// TwinCAT 3 PLC project PLC1
// ProgramVersion: 3.1.4022.2
// libraries:
//   ERS_CO2 Payload Decoder, * (PXL-Tech)
//   MSC1608 Payload Decoder, * (PXL-Tech)
//   Tc2_BABasic, * (Beckhoff Automation GmbH)
//   Tc2_EnOcean, * (Beckhoff Automation GmbH)
//   Tc2_Standard, * (Beckhoff Automation GmbH)
//   Tc2_System, * (Beckhoff Automation GmbH)
//   Tc2_TcpIp, * (Beckhoff Automation GmbH)
//   Tc2_Utilities, * (Beckhoff Automation GmbH)
//   Tc3_JsonXml, * (Beckhoff Automation GmbH)
//   Tc3_Module, * (Beckhoff Automation GmbH)
//   VisuSymbols,3.5.10.0,System
// project tree:
//   DUTs/ ST_Gwrx.TcDUT, ST_MoteTx.TcDUT, ST_UserData.TcDUT
//   / GlobalTextList.TcGTLO, PlcTask.TcTTO (not stored), Visualization Manager.TcVMO (not stored), VISU_TASK.TcTTO
//   GVLs/ GVL1.TcGVL
//   POUs/ Decoder.TcPOU, DecoderCO2.TcPOU, EnOcean.TcPOU, Json_XML.TcPOU, Lichtsturing.TcPOU, MAIN.TcPOU, Beamercontrol.TcPOU, Tcp_ip.TcPOU
//   VISUs/ Visualization.TcVIS, Visualization_1.TcVIS
// real-time tasks:
//   TASK PlcTask: cycle T#10ms, priority 6, ADS port 350
//   TASK VISU_TASK: cycle T#200000us, priority 30, ADS port 351
//   TASK Standard: cycle T#5ms, priority 20, ADS port 352
// I/O:
//   DEVICE Device 1 (EtherCAT), AmsNetId 5.52.70.129.2.1
//     Term 7 (EK1200) [EK1200-5000 EtherCAT Power supply (2A E-Bus)]
//       Term 8 (EL1008) [EL1008 8Ch. Dig. Input 24V, 3ms]
//       Term 9 (EL2008) [EL2008 8Ch. Dig. Output 24V, 0.5A]
//       Term 10 (EL3062) [EL3062 2Ch. Ana. Input 0-10V]
//       Term 11 (EL4002) [EL4002 2Ch. Ana. Output 0-10V, 12bit]
//       Term 12 (EK1122) [EK1122 2 port EtherCAT junction]
//         Box 13 (BK1150)
//   DEVICE Device 3 (RT-Ethernet Protocol), AmsNetId 5.52.70.129.4.1
//   DEVICE Device 2 (NOV-DP-RAM)
// variable links:
//   EnOcean_Sample_CX9020/EnOcean_Sample_CX9020 Instance <-> Device 1 (EtherCAT)/Term 7 (EK1200)/Term 12 (EK1122)/Box 13 (BK1150)
//     Standard Inputs/.st6581Input/CNODE <-> Term 2 (KL6581)/Channel 1/Input CNODE
//     Standard Inputs/.st6581Input/DB{0..3} <-> Term 2 (KL6581)/Channel 1/Input DB{0..3}  (4 links)
//     Standard Inputs/.st6581Input/ID{0..3} <-> Term 2 (KL6581)/Channel 1/Input ID{0..3}  (4 links)
//     Standard Inputs/.st6581Input/ORG <-> Term 2 (KL6581)/Channel 1/Input ORG
//     Standard Inputs/.st6581Input/STATUS <-> Term 2 (KL6581)/Channel 1/Input STATUS
//     Standard Inputs/.st6581Input/nStatus <-> Term 2 (KL6581)/Channel 1/Status
//     Standard Outputs/.st6581Output/CNODE <-> Term 2 (KL6581)/Channel 1/Output CNODE
//     Standard Outputs/.st6581Output/DB{0..3} <-> Term 2 (KL6581)/Channel 1/Output DB{0..3}  (4 links)
//     Standard Outputs/.st6581Output/ID{0..3} <-> Term 2 (KL6581)/Channel 1/Output ID{0..3}  (4 links)
//     Standard Outputs/.st6581Output/ORG <-> Term 2 (KL6581)/Channel 1/Output ORG
//     Standard Outputs/.st6581Output/STATUS <-> Term 2 (KL6581)/Channel 1/Output STATUS
//     Standard Outputs/.st6581Output/nControl <-> Term 2 (KL6581)/Channel 1/Control

CONFIGURATION PLC1
    RESOURCE PLC ON TwinCAT3
        TASK VISU_TASK(INTERVAL := T#200000us, PRIORITY := 30);
        PROGRAM VisuElems_Visu_Prg WITH VISU_TASK : VisuElems.Visu_Prg;
    END_RESOURCE
END_CONFIGURATION

// ---- DUTs/ST_Gwrx.TcDUT
TYPE ST_Gwrx :
STRUCT
	TimeRec	: STRING;//DATE_AND_TIME ;
	Chan : DINT ;
	Rfch : DINT ;
	Rssi : DINT ;
	Lsnr : REAL ;
END_STRUCT
END_TYPE

// ---- DUTs/ST_MoteTx.TcDUT
TYPE ST_MoteTx :
STRUCT
	Freq	: DINT ;
	Modu	: STRING(20);
	Datr	: STRING(20);
	Codr	: STRING(20);
END_STRUCT
END_TYPE

// ---- DUTs/ST_UserData.TcDUT
TYPE ST_UserData :
STRUCT
	SeqNo	: DINT;
	Port	: DINT;
	Payload	: STRING;
	Payload2: DINT;
	MoteTx	: ST_MoteTx;
	Gwrx : ST_Gwrx;
END_STRUCT
END_TYPE

// ---- GVLs/GVL1.TcGVL
VAR_GLOBAL
	
//lichtsturing
LichtenRAAMKANT AT %Q*: BOOL;
LichtenDEURKANT AT %Q*: BOOL;

AanwezigheidsdetectorRAAMKANT AT %I*: BOOL;
AanwezigheidsdetectorDEURKANT AT %I*: BOOL;

LichtsterkteDEUR AT %I*: INT;
LichtsterkteDEUR2 AT %I*: INT;
LichtsterkteBORD AT %I*: INT;
lichtsterkteBORD2 AT %I*: INT;
LINKERKNOP AT %I* : BOOL;
RECHTERKNOP AT %I* : BOOL;


//beamer & projectorschermsturing

BeamerAANKNOP AT %I* : BOOL;
BeamerUITKNOP AT %I* : BOOL;
Projectorscherm AT %Q* : BOOL;



socketconnectknop AT %I* : BOOL;
socketsendknop AT %I* : BOOL;



//raamsturing


stKL6581            : STR_KL6581;


//Lora
	sDatastring: STRING(500);
	
	Moteeui			: STRING;
	Appeui			: STRING;
	UserData		: ST_UserData;
	PayloadDecoded	: STRING;

	PayloadLength	: DINT;
	PayloadData		: ARRAY[1..100] OF BYTE;
	NullByte		: BYTE := 0;


END_VAR

// ---- POUs/Lichtsturing.TcPOU
PROGRAM Lichtsturing

 VAR PERSISTENT
	relaisstandDEUR : BOOL := FALSE;
 	relaisstandRAAM : BOOL := FALSE;
 
 
 END_VAR
 
 
VAR
	timer1: TOF;
	timer2: TOF;
	TP1: TP;
	TP2 : TP;
	TP3 : TP;
	TP4 : TP;
	TP5 :TP;
	TP6 : TP;
	
	bewegingraam : BOOL;
	bewegingdeur : BOOL;
	relaisstandDEUR_nieuw : BOOL := FALSE;
	lichtstand2 : BOOL;
	Lichtstand_Prev2: BOOL;
	Lichtstand_Prev: BOOL;
	LichtstatusDEUR : BOOL;
	LichtstatusBORD : BOOL;
	
	

	TONBOOL: BOOL;
	TON1: TON;
	rtrigger: R_TRIG;
	rtrigger2: R_TRIG;
	rtrigger3: R_TRIG;
	rtrigger4: R_TRIG;
	LINKERKNOPULS: BOOL;
	RECHTERKNOPPULS: BOOL;
	
	lichtsterktedeurBerekening: INT := 30000;
	lichtsterkteraamBerekening: INT := 15000;
	fblicht: FB_Light;
	fblicht2 : FB_light;
	relaisstandraam_nieuw: BOOL;
END_VAR

timer1(IN:=gvl1.AanwezigheidsdetectorRAAMKANT, PT:= T#300S, Q=>bewegingraam, ET=> );
timer2(IN:=gvl1.AanwezigheidsdetectorDEURKANT, PT:= T#300S, Q=>bewegingdeur , ET=> );



fblicht(bOn:= (LichtsterkteDEUR + LichtsterkteDEUR2 < lichtsterktedeurBerekening AND bewegingdeur = TRUE), 
bOff:= NOT (LichtsterkteDEUR + LichtsterkteDEUR2 < lichtsterktedeurBerekening AND bewegingdeur = TRUE), 
bToggle:=RECHTERKNOP, bLight=> relaisstandDEUR_nieuw);

IF (relaisstandDEUR = NOT relaisstandDEUR_nieuw) THEN
	TP2.IN := TRUE;
	relaisstandDEUR := relaisstandDEUR_nieuw;
ELSE
	TP2.IN := FALSE;
END_IF


TP2( PT:=T#50MS , Q => GVL1.LichtenDEURKANT);


fblicht2(bOn:= (LichtsterkteBORD + lichtsterkteBORD2 < lichtsterkteraamBerekening AND bewegingraam = TRUE), 
bOff:= NOT (LichtsterkteBORD + lichtsterkteBORD2 < lichtsterkteraamBerekening AND bewegingraam = TRUE), 
bToggle:=LINKERKNOP, bLight=> relaisstandraam_nieuw);

IF (relaisstandraam = NOT relaisstandraam_nieuw) THEN
	TP1.IN := TRUE;
	relaisstandraam := relaisstandraam_nieuw;
ELSE
	TP1.IN := FALSE;
END_IF


TP1( PT:=T#50MS , Q => GVL1.LichtenRAAMKANT);

END_PROGRAM

// ---- POUs/Decoder.TcPOU
PROGRAM Decoder
VAR
 	FB_Decoder : MCS1608_Payload_Decoder;
    //GenSens
 	Status     			:BYTE;      // Content Depends on Message ID == for future use
	BaromBar			:REAL;      // Air Pressure in mBar
	Temp1   			:REAL;     	// in 0,01 degC
	Humidity   			:BYTE;      // Relative Humidity in %
	LevelX     			:SINT;      // Inverse Sinus of Spirit Level in Deg X-Direction -128 = -90 Degr .. +127 = +90 Degr
	LevelY     			:SINT;      // Inverse Sinus of Spirit Level in Deg Y-Direction -128 = -90 Degr .. +127 = +90 Degr
	LevelZ     			:SINT;      // Inverse Sinus of Spirit Level in Deg Z-Direction -128 = -90 Degr .. +127 = +90 Degr
	VibAmp     			:USINT;     // Amplitude of Vibration Detected == Future
	VibFreq    			:USINT;     // Approx. Frequency of Vibration Detected in Hz == Future



	//Tracking
	Start				:BOOL;// Start Message
	Moving				:BOOL;// Object Moving
	Stop				:BOOL;// Object Stopped
	Vibr				:BOOL;// Vibration Detected
	Temp2				:REAL;// Temperature in 0,01 degC
	GPSFixAge			:BYTE;// bit 0..7 = Age of last GPS Fix in Minutes,
	SatCnt_HiLL			:BYTE;// bit 0..4 = SatInFix, bit5 Latitude 25 bit 6,7 = Longitude 25,26
	Lat					:REAL;
	Lon					:REAL;
	
	//Alarm
	GravRotAl		:BOOL;	// Gravity Rotation Detected
	MagRot			:BOOL;	// Magnetic Rotation Detected
	MotAlarm		:BOOL;	// Motion Alarm Detected
	GeoFenceAl		:BOOL;	// GeoFence Violation Detected
	VibrAl			:BOOL;	// Vibration Alarm Detected
	ShockAl			:BOOL;	// Shock Alarm (future use)
	DigIn1Al		:BOOL;	// Digin1 Alarm Detected
	DigIn2Al		:BOOL;	// Digin2 Alarm Detected
	Temp			:REAL;	// Temperature in 0,01 Celcius
	Hum				:BYTE;	// Relative Humidity in %
	BaromBar2		:REAL;	// Air Pressure in Mbar
	
	Alarm1 : Alarm; 
END_VAR

FB_Decoder(dataString := PayloadDecoded);

CASE FB_Decoder.MsgID OF 
	FB_Decoder.ID_Tracking:
		//Start := FB_Decoder.Tracking.Start;
		Moving := FB_Decoder.Tracking.Moving;
		Stop := FB_Decoder.Tracking.Stop;
		Vibr := FB_Decoder.Tracking.Vibr;
		Temp2 := FB_Decoder.Tracking.Temp;
		GPSFixAge := FB_Decoder.Tracking.GPSFixAge;
		SatCnt_HiLL	:= FB_Decoder.Tracking.SatCnt_HiLL;
		Lat	:= FB_Decoder.Tracking.Lat;
		Lon	:= FB_Decoder.Tracking.Lon;
	FB_Decoder.ID_Alarm:
		Alarm1.MotAlarm := FB_Decoder.Alarm.MotAlarm;
	FB_Decoder.ID_GenSens:
		Status := FB_Decoder.GenSens.Status;
		BaromBar := FB_Decoder.GenSens.BaromBar;
		Temp := FB_Decoder.GenSens.Temp;
		Humidity := FB_Decoder.GenSens.Humidity;
		LevelX := FB_Decoder.GenSens.LevelX;
		LevelY := FB_Decoder.GenSens.LevelY;
		LevelZ := FB_Decoder.GenSens.LevelZ;
		VibAmp := FB_Decoder.GenSens.VibAmp;
		VibFreq := FB_Decoder.GenSens.VibFreq;
END_CASE

END_PROGRAM

// ---- POUs/DecoderCO2.TcPOU
PROGRAM DecoderCO2
VAR
	FB_Decoder : ERS_CO2_PayloadDecoder;
	
	Temperature 	: REAL;		//Temp -3276.8°C - 3276.7°C
	Humidity 		: BYTE;		//Humidity 0-100%
	X 				: REAL;		//Acceleration X -128 --> 127 +/-63 = 1G
	Y 				: REAL;		//Acceleration Y -128 --> 127 +/-63 = 1G
	Z 				: REAL;		//Acceleration Z -128 --> 127 +/-63 = 1G
	Light 			: WORD; 	//Light 0 - 65535 Lux
	Motion 			: BYTE;		//No of motion 0-255
	Co2				: WORD;		//Co2 0-65535 ppm 
	Vdd				: WORD;		//VDD 0-65535mV
	Analog1			: WORD;		//VDD 0-65535mV
	Lat				: DWORD;	//Latitude binary
	Lon				: DWORD;	//Longitude binary
	Pulse1			: WORD;		//Relative pulse count
	pulseAbs		: DWORD;	//no 0 - 0xFFFFFFFF
	ExternalTemp	: REAL;		//External temp -3276.5C-->3276.5C
	Digital			: BYTE;		//Value 1 or 0
	Distance		: WORD;		//Distance in mm
	AccMotion		: BYTE;		//Number of vibration/motion
	IrInternalTemp	: REAL;		//Internal temp -3276.5C - 3276.5C
	IrExternalTemp	: REAL;		//External temp -3276.5C - 3276.5C
	Occupancy		: BYTE;		//Data
	Waterleak		: BYTE;		//Data 0-255
	Pressure		: REAL;		//Pressure data(hPa)
	SoundPeak		: BYTE;		//Sound peak
	SoundAvg		: BYTE;		//Sound average
	Pulse2			: WORD;		//0 - 0xFFFF
	PulseAbs2		: DWORD;	//no 0 - 0xFFFFFFFF
	Analog2			: WORD;		//Voltage in mV
	ExternalTemp2	: REAL;		//External temp2 -3276.5C - 3276.5C
END_VAR

FB_Decoder(dataString := PayloadDecoded);

		Temperature 	:= FB_Decoder.Temperature;
		Humidity 		:= FB_Decoder.Humidity;
		X 				:= FB_Decoder.X;
		Y 				:= FB_Decoder.Y;
		Z 				:= FB_Decoder.Z;
		Light 			:= FB_Decoder.Light;		
		Motion 			:= FB_Decoder.Motion;
		Co2				:= FB_Decoder.Co2; 
		Vdd				:= FB_Decoder.Vdd;
		Analog1			:= FB_Decoder.Analog1;
		Lat				:= FB_Decoder.Lat;
		Lon				:= FB_Decoder.Lon;
		Pulse1			:= FB_Decoder.Pulse1;
		pulseAbs		:= FB_Decoder.pulseAbs;
		ExternalTemp	:= FB_Decoder.ExternalTemp;
		Digital			:= FB_Decoder.Digital;
		Distance		:= FB_Decoder.Distance;
		AccMotion		:= FB_Decoder.AccMotion;
		IrInternalTemp	:= FB_Decoder.IrInternalTemp;
		IrExternalTemp	:= FB_Decoder.IrExternalTemp;
		Occupancy		:= FB_Decoder.Occupancy;
		Waterleak		:= FB_Decoder.Waterleak;
		Pressure		:= FB_Decoder.Pressure;
		SoundPeak		:= FB_Decoder.SoundPeak;
		SoundAvg		:= FB_Decoder.SoundAvg;
		Pulse2			:= FB_Decoder.Pulse2;
		PulseAbs2		:= FB_Decoder.PulseAbs2;
		Analog2			:= FB_Decoder.Analog2;
		ExternalTemp2	:= FB_Decoder.ExternalTemp2;

END_PROGRAM

// ---- POUs/EnOcean.TcPOU
PROGRAM EnOcean

VAR
	
FBRECEX: FB_Rec_Teach_In_Ex;


rxD: FB_KL6581;
fbkl6581: FB_KL6581;
	
stKL6581_in AT %I* : KL6581_Input;
stKL6581_out AT %Q* : KL6581_Output; 


testvar2: INT;
	generic1: FB_Rec_1BS;
	generic2: FB_Rec_1BS;
END_VAR



VAR_INPUT 
	//84246605
	//84246441
//fbkl6581
bInit             : BOOL;
nIdx              : USINT := 2;


//FBRECEX
	
bStart            : BOOL;
byNode            : BYTE;
str_KL6581        : STR_KL6581;
DeviceID : DWORD := 0;
testvar : INT := 0;

dw_ID                  : DWORD;

END_VAR



VAR_OUTPUT
	

bReady            : BOOL;
bBusy             : BOOL;
bError            : BOOL;
iErrorID          : E_KL6581_Err;

	

	
bLearnType        : BOOL;
by_Node           : BYTE;

str_Teach_In      : STR_Teach;
bReceive          : BOOL := TRUE;
bReceive2         : BOOL := TRUE;


raam1open          : BOOL;
raam1gesloten          : BOOL;
bLRN            : BOOL;

raam2open         : BOOL;
raam2gesloten         : BOOL;
bLRN2           : BOOL;


END_VAR


fbkl6581(
	bInit:= TRUE , 
	nIdx:= nIdx, 
	bReady=> bReady, 
	bBusy=> bBusy, 
	bError=> bError, 
	iErrorID=> iErrorID, 
	str_KL6581=> str_KL6581, 
	
	stKL6581_in:= stKL6581_in, 
	stKL6581_out:= stKL6581_out);
	
	

FBRECEX(
	bStart:= TRUE, 
	byNode:= 0,
	str_KL6581:= str_KL6581, 
	bLearnType=> , 
	by_Node=>by_node, 
	dw_ID=>DeviceID, 
	str_Teach_In=> str_Teach_In , );
	//bReceive=>bReceive );
	
	
	generic1(
	str_KL6581:= str_KL6581  , 
	byNode:= 0, 
	dw_ID:= 84246605, 
	bOpen=> raam1open, 
	bClose=> raam1gesloten, 
	bLRN=> bLRN2, 
	by_Node=> , 
	bReceive=>bReceive );
	
	generic2(
	str_KL6581:= str_KL6581  , 
	byNode:= 0, 
	dw_ID:= 84246441, 
	bOpen=> raam2open, 
	bClose=> raam2gesloten, 
	bLRN=> bLRN, 
	by_Node=> , 
	bReceive=> bReceive2);

END_PROGRAM

// ---- POUs/Json_XML.TcPOU
PROGRAM Json_XML
VAR
	
	//sJsontest		: STRING(500) := '{"rx": {"moteeui": "00-59-ac-00-00-15-10-ee", "appeui": "0000000000000000", "userdata": {"seqno": 122, "port": 1, "payload": "MDIwMDA1YWUwOTdhMzYwMDAwZmEwMDAwMDAwMDAwMDA=", "motetx": {"freq": 868300000, "modu": "LoRa", "datr": "SF8BW125", "codr": "4/5"}}, "gwrx":  [{"time": "2017-10-17 12:34:53", "chan": 4, "rfch": 0, "rssi": -34, "lsnr": 11.800000000000001}]}}';	
	//sJsontest		: STRING(500) := '{"rx": {"moteeui": "00-59-ac-00-00-15-10-ee", "appeui": "0000000000000000", "userdata": {"seqno": 122, "port": 1, "payload": "MDIwMDA1YWUwOTdhMzYwMDAwZmEwMDAwMDAwMDAwMDA=", "motetx": {"freq": 868300000, "modu": "LoRa", "datr": "SF8BW125", "codr": "4/5"}}, "gwrx": [{"time": "2017-10-17 12:34:53", "chan": 4, "rfch": 0, "rssi": -34, "lsnr": 11.800000000000001}]}}';	
	
	x : DINT;
	g : STRING;
	fbJson			: FB_JsonDomParser;
	JsonDoc			: SJsonValue;
	Json_St1		: SJsonValue;
	JSon_St2		: SJsonValue; 
	JSon_St3		: SJsonValue;
	JSon_St4		: SJsonValue;
	JSon_St5		: SJsonValue;
	JSon_St6		: SJsonValue;
	Stringdata		: STRING;
	
	i: INT;
END_VAR

FOR i := 0 TO 498 DO										//Forloop doorloop elk teken appart
	IF sDatastring[i] = 91 OR sDatastring[i] = 93 THEN		//ALs er een vierkante haak  voor komt
		sDatastring[i] := 32;								//Zal het door een spatie gewijzigd worden
	END_IF
END_FOR

JsonDoc := fbJson.ParseDocument(sDatastring);

// rx
Json_St1 := fbJson.FindMember(jsonDoc, 'rx');			

	// moteeui 
	JSon_St2 := fbJson.FindMember(Json_St1, 'moteeui');
	Moteeui := fbJson.GetString(JSon_St2);

	// appeui	
	JSon_St2 := fbJson.FindMember(Json_St1, 'appeui');
	Appeui := fbJson.GetString(JSon_St2);

	// userdata
	JSon_St2 := fbJson.FindMember(Json_St1, 'userdata');

		// seqno
		JSon_St3 := fbJson.FindMember(Json_St2, 'seqno');
		UserData.SeqNo := fbJson.GetInt(JSon_St3);

		// port
		JSon_St3 := fbJson.FindMember(Json_St2, 'port');
		UserData.Port := fbJson.GetInt(JSon_St3);

		// payload
		JSon_St3 := fbJson.FindMember(Json_St2, 'payload');
		UserData.Payload := fbJson.GetString(JSon_St3);
		PayloadLength:= fbJson.GetBase64(JSon_St3, ADR(PayloadData), SIZEOF(PayloadData));
		Memcpy(ADR(PayloadDecoded), ADR(PayloadData), PayloadLength);
		Memcpy(ADR(PayloadDecoded)+PayloadLength, adr(NullByte), 1);

		// motetx
		JSon_St3 := fbJson.FindMember(Json_St2, 'motetx');

			// freq
			JSon_St4 := fbJson.FindMember(Json_St3, 'freq');
			UserData.MoteTx.Freq := fbJson.GetInt(JSon_St4);

			// modu
			JSon_St4 := fbJson.FindMember(Json_St3, 'modu');
			UserData.MoteTx.Modu := fbJson.GetString(JSon_St4);

			// datr
			JSon_St4 := fbJson.FindMember(Json_St3, 'datr');
			UserData.MoteTx.Datr := fbJson.GetString(JSon_St4);

			// codr
			JSon_St4 := fbJson.FindMember(Json_St3, 'codr');
			UserData.MoteTx.Codr := fbJson.GetString(JSon_St4);

		// gwrx
		JSon_St5 := fbJson.FindMember(Json_St1, 'gwrx');
		Stringdata := fbJson.GetString(JSon_St5);

		// seqno
		JSon_St6 := fbJson.FindMember(Json_St5, 'time');
		UserData.gwrx.TimeRec  := fbJson.GetString(JSon_St6);

END_PROGRAM

// ---- POUs/MAIN.TcPOU
PROGRAM MAIN
VAR
END_VAR

Lichtsturing();
EnOcean();
Beamercontrol();
Tcp_ip();

END_PROGRAM

// ---- POUs/Beamercontrol.TcPOU
PROGRAM Beamercontrol



VAR
	
	fbsocketsend: FB_SocketSend;
	bconnect AT %I* : BOOL;
	test : int;
	clientserver: FB_ClientServerConnection;


	
	Beamerstand: LINT;
END_VAR


VAR_INPUT

       
nMode           : DWORD := 16#8000000;



 
BeamerON    : LINT := 16#020000000002;


BeamerOFF 	: LINT := 16#020100000003;
					  

beamerINPUTCHANGE : LINT :=16#020300000201060E;


	
	 


      	sSrvNetId       : T_AmsNetId := '5.52.70.129.1.1';
	  
        sRemoteHost     : STRING(15) := '192.168.0.102';
        nRemotePort     : UDINT := 7142;
        bExecute                : BOOL;
        tTimeout                : TIME := T#45S;
		tReconnect      : TIME := T#45S;(*!!!*)
		

//socketsend       
               
        cbLen           : UDINT;                        
        pSrc            : DWORD;    
		            
           
END_VAR  

VAR_OUTPUT
        bBusy           : BOOL;
        bError          : BOOL;
        nErrId          : UDINT;
		nErrId2          : UDINT;
        hSocket        : T_HSOCKET;
		eState          : E_SocketConnectionState := eSOCKET_DISCONNECTED;
		
	
END_VAR

clientserver(
	sSrvNetID:= '', 
	nMode:=CONNECT_MODE_ENABLEDBG , 
	sRemoteHost:= sremoteHost , 
	nRemotePort:= nremoteport, 
	bEnable:= bconnect, 
	tReconnect:= tReconnect, 
	bBusy=> bBusy, 
	bError=> berror,
	nErrId=>nErrId , 
	hSocket=>hsocket , 
	eState=> eState);
	
	IF BeamerAANKNOP = TRUE THEN
		bExecute := TRUE;
		Beamerstand := BeamerON;
ELSE
	IF BeamerUITKNOP = TRUE THEN
		bExecute := TRUE;
		Beamerstand := BeamerOFF;
	ELSE
		bExecute := FALSE;
		Beamerstand := 0;
	END_IF
	END_IF
	
fbsocketsend(
	sSrvNetId:='' , 
	hSocket:= clientserver.hSocket, 
	cbLen:= 50, 
	pSrc:= ADR(Beamerstand), 
	bExecute:= bexecute , 
	tTimeout:=tTimeout , 
	bBusy=> bBusy , 
	bError=> bError, 
	nErrId=> nErrId2);

END_PROGRAM

// ---- POUs/Tcp_ip.TcPOU
PROGRAM Tcp_ip
VAR
	bConnect: BOOL;
	bRecieve: BOOL;
	FB_create: FB_SocketUdpCreate;
	FB_Recieve: FB_SocketUdpReceiveFrom;
	FB_close: FB_SocketClose;
	data : ARRAY[0..500] OF BYTE;
END_VAR

FB_create(
	sSrvNetId:= , 							//Lokaal netwerk (mag leeg blijven)
	sLocalHost:= '192.168.0.104', 			//Eigen ip van de PC en ingesteld in de gateway
	nLocalPort:= 811,						//Ingesteld op de gateway
	bExecute:= bConnect,					//Trigger voor functieblok
	tTimeout:= T#45S);
	

FB_Recieve(
	sSrvNetId:= , 									//Lokaal netwerk (mag leeg blijven)
	hSocket:= FB_create.hSocket,					 
	cbLen:= SIZEOF(data), 							//Kijkt naar de lengte van het bericht
	pDest:= ADR(data), 								//Plaat waar de het bericht wordt opgeslaan
	bExecute:= NOT FB_recieve.bBusy AND bRecieve, 	//Trigger voor functieblok
	tTimeout:= T#45S);
	
FB_close(
	sSrvNetId:= , 							//Lokaal netwerk (mag leeg blijven)
	hSocket:= FB_create.hSocket, 			
	bExecute:= NOT bConnect, 				//Sluiten van de connectie 
	tTimeout:= T#45S);
	
IF FB_Recieve.nRecBytes > 0 THEN 										//Dit gebuert op het moment dat er data binnenkomt
	memcpy(ADR(sDatastring),ADR(data),FB_Recieve.nRecBytes);			//Het bericht zal worden opgeslaan in Datastring
	memcpy(ADR(sDatastring) + FB_Recieve.nRecBytes,ADR(NullByte),1);	//Nullbyte word gedetecteerd stoppen met bericht plaatsen
	Json_XML();															//Oproepen POU Json_XML - MOET hier anders bluescreen
	Decoder();
	DecoderCO2();															//Oproepen POU Decoder  - MOET hier anders bluescreen
END_IF

END_PROGRAM

// ---- GlobalTextList.TcGTLO
TEXTLIST GlobalTextList
  820 = 'Bar : %d'
  42 = 'Beamer OFF'
  198 = 'Beamer ON'
  817 = 'Close'
  831 = 'Conection'
  492 = 'Connect'
  830 = 'Create'
  833 = 'Datum/Tijd : %s'
  787 = 'Deurkant'
  828 = 'Error'
  822 = 'Humidity : %d %'
  823 = 'Level x : %d'
  824 = 'Level y : %d'
  825 = 'Level z : %d'
  818 = 'Mesage ID : %d'
  816 = 'Payload : %s'
  774 = 'Raamkant'
  815 = 'Recieve'
  829 = 'Sensor ID : %s'
  819 = 'Status : %d'
  821 = 'Temp : %.2f °c'
  832 = 'Type sensor : '
  826 = 'VibAmp : %d'
  827 = 'VidFreq : %d'
END_TEXTLIST

// ---- VISUs/Visualization.TcVIS
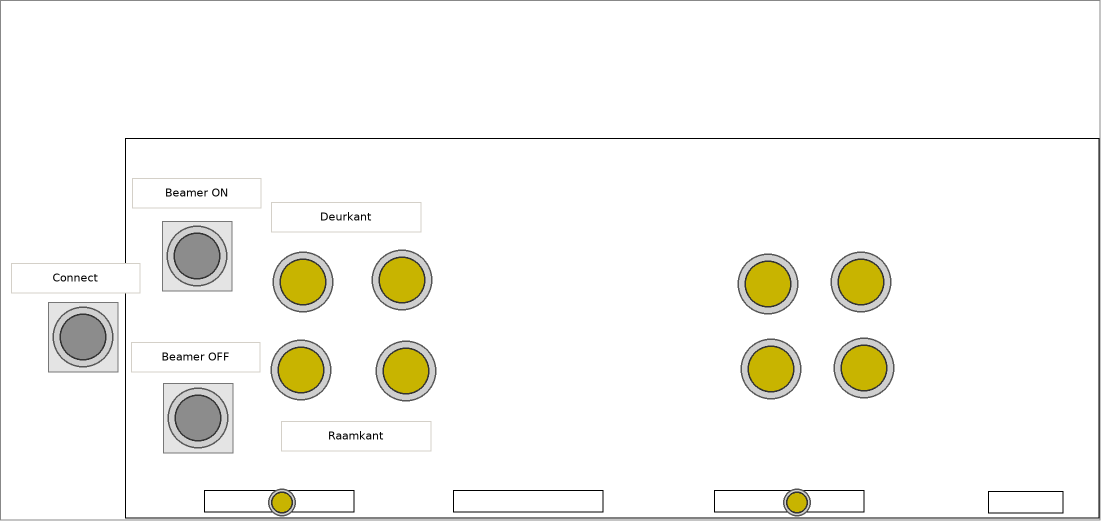
VISUALIZATION Visualization  // 1101x521
    Rectangle (125,138 974x380)
    Lamp1 (268,247 70x70), variable: Lichtsturing.relaisstandDEUR, style: Lamp-Lamp1-Yellow
    Lamp1 (367,245 70x70), variable: Lichtsturing.relaisstandDEUR, style: Lamp-Lamp1-Yellow
    Lamp1 (733,249 70x70), variable: Lichtsturing.relaisstandDEUR, style: Lamp-Lamp1-Yellow
    Lamp1 (826,247 70x70), variable: Lichtsturing.relaisstandDEUR, style: Lamp-Lamp1-Yellow
    Lamp1 (266,335 70x70), variable: Lichtsturing.relaisstandRAAM, style: Lamp-Lamp1-Yellow
    Lamp1 (371,336 70x70), variable: Lichtsturing.relaisstandRAAM, style: Lamp-Lamp1-Yellow
    Lamp1 (736,334 70x70), variable: Lichtsturing.relaisstandRAAM, style: Lamp-Lamp1-Yellow
    Lamp1 (829,333 70x70), variable: Lichtsturing.relaisstandRAAM, style: Lamp-Lamp1-Yellow
    Rectangle (204,490 150x22)
    Rectangle (453,490 150x22)
    Rectangle (714,490 150x22)
    Rectangle (988,491 75x22)
    Lamp1 (266,486 32x33), variable: EnOcean.raam2open, style: Lamp-Lamp1-Yellow
    Lamp1 (781,486 32x33), variable: EnOcean.raam1open, style: Lamp-Lamp1-Yellow
    Textfield (271,202 150x30), "Deurkant"
    Textfield (281,421 150x30), "Raamkant"
    PushSwitch (162,221 70x70), variable: BeamerAANKNOP, behaviour: TOGGLE, style: Switch-PushSwitch-Gray
    Textfield (132,178 129x30), "Beamer ON"
    PushSwitch (163,383 70x70), variable: BeamerUITKNOP, behaviour: TOGGLE, style: Switch-PushSwitch-Gray
    Textfield (131,342 129x30), "Beamer OFF"
    PushSwitch (48,302 70x70), variable: Beamercontrol.bconnect, behaviour: TOGGLE, style: Switch-PushSwitch-Gray
    Textfield (11,263 129x30), "Connect"
END_VISUALIZATION

// ---- VISUs/Visualization_1.TcVIS
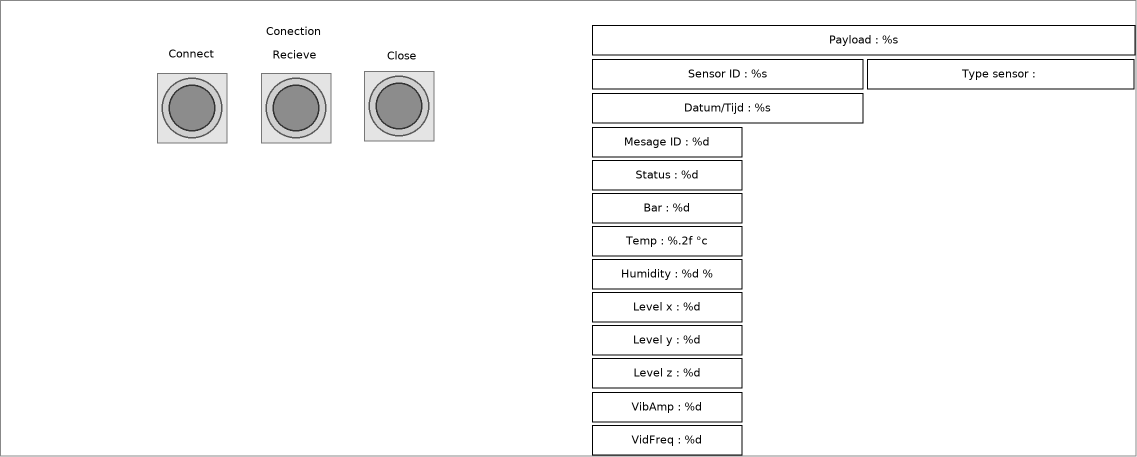
VISUALIZATION Visualization_1  // 1137x457
    PushSwitch (157,73 70x70), variable: Tcp_ip.bConnect, behaviour: TOGGLE, style: Switch-PushSwitch-Gray
    Label (156,39 71x30), "Connect"
    PushSwitch (261,73 70x70), variable: Tcp_ip.bRecieve, behaviour: TOGGLE, style: Switch-PushSwitch-Gray
    Label (261,40 67x30), "Recieve"
    Rectangle (592,25 543x30), "Payload : %s", text variable: PayloadDecoded
    PushSwitch (364,71 70x70), variable: Tcp_ip.FB_close.bExecute, behaviour: TOGGLE, style: Switch-PushSwitch-Gray
    Label (369,41 66x30), "Close"
    Rectangle (592,127 150x30), "Mesage ID : %d", text variable: Decoder.FB_Decoder.MsgID
    Rectangle (592,160 150x30), "Status : %d", text variable: Decoder.Status
    Rectangle (592,193 150x30), "Bar : %d", text variable: Decoder.BaromBar
    Rectangle (592,226 150x30), "Temp : %.2f °c", text variable: Decoder.Temp
    Rectangle (592,259 150x30), "Humidity : %d %", text variable: Decoder.Humidity
    Rectangle (592,292 150x30), "Level x : %d", text variable: Decoder.LevelX
    Rectangle (592,325 150x30), "Level y : %d", text variable: Decoder.LevelY
    Rectangle (592,358 150x30), "Level z : %d", text variable: Decoder.LevelZ
    Rectangle (592,392 150x30), "VibAmp : %d", text variable: Decoder.VibAmp
    Rectangle (592,425 150x30), "VidFreq : %d", text variable: Decoder.VibFreq
    Rectangle (592,59 271x30), "Sensor ID : %s", text variable: Moteeui
    Label (165,17 257x29), "Conection"
    Rectangle (867,59 267x30), "Type sensor :"
    Rectangle (592,93 271x30), "Datum/Tijd : %s", text variable: UserData.Gwrx.TimeRec
END_VISUALIZATION
